(* CoDeSys 2.3 export: GVL.EXP *)

(* Global variable list: Global_Variables *)
VAR_GLOBAL
	H_com: UINT;		(*час реального времени*)
	M_com: UINT;		(*минуты реального времени*)
	S_com: UINT;		(*секунды реального времени*)
	(*Версия ПО*)
	VERSION_M:WORD	:= 2;
	VERSION_L:WORD 	:= 0;

	INITIAL:BOOL:=TRUE;

	DI_BUF: WORD;
	AI_BUF : ARRAY [0..3] OF REAL;
	CountDI : INT :=8;
	CountDO:INT := 32;
	CountAI : INT :=4;
	DI_ARRAY : ARRAY [0..7] OF tDI; (*Массив DI*)
	DO_ARRAY : ARRAY[0..31] OF tDO; (*массив DO*)
	AI_ARRAY : ARRAY[0..3] OF tAI; (*массив AI*)
	DozVars : ARRAY[0..1] OF tDoz;	(*массив переменных дозаторов 0 - ес, 1 - ph*)
	Rasp_ARRAY : ARRAY [0..31] OF tRasp;

	global_auto_manual	: BOOL;	(*глобальны авто/ручн режим*)
END_VAR
